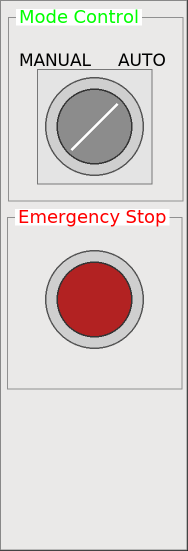
VISUALIZATION SysPanel  // 188x551
    Rectangle (0,0 188x551)
    GroupBox (8,9 175x192), "Mode Control"
        Label (4,36 86x30), "MANUAL"
        Label (105,36 58x30), "AUTO"
        RotarySwitch (29,60 115x115), variable: gvlMotion.manualMode, behaviour: TOGGLE, style: Switch-RotarySwitch-Gray
    GroupBox (7,209 175x180), "Emergency Stop"
        Lamp1 (30,33 115x115), tooltip "!", variable: TRUE, style: Lamp-Lamp1-Red
END_VISUALIZATION

(* stored: Version 1.1.0.1, ProductVersion 3.1.4024.12
   Visu SysPanel: Id {4682090b-b4c5-4b3a-b968-10e30293b3ef} *)
